ABB RobotStudio station: Robot_1530ID (task 1).rsstn

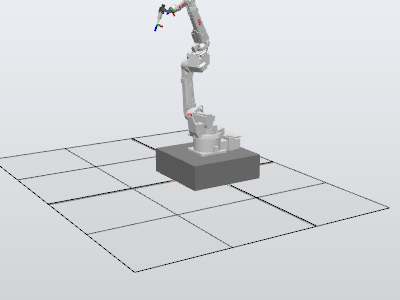
Station Robot_1520ID (frist class) (saved by RobotStudio 22.3.10141.1)
Controller Controller17, task T_ROB1: task frame (RAPID world) sits at (0, 0, 290) mm in the station
Controller Controller17
  mechanical unit ROB_1: IRB1520ID_4_150__02, 6 joints, base frame (0, 0, 0) mm
Layout (positions relative to the parent item):
  - IRB1520ID_4_150__02 [mechanism, from Robots\IRB1520ID_4_150_G_02.rslib] at (0, 0, 290) mm; joint values [0.1655, 0.0623, -1.1863, -0.1436, 1.6527, 0.0715] (rad or m)
  - Part_1_2 [part, from Robotics 7020\Cement Base.rslib] at (-450, -450, 0) mm
  - MyTool [mechanism, from Training Objects\myTool.rslib] at (497.52, 54.16, 1970.29) mm, rotated rx 180 ry 60 rz -180 deg
Attachment: MyTool is attached to IRB1520ID_4_150__02 / Link6
Targets, tools, work objects and paths stored in the station, written as RAPID:
! task T_ROB1
MODULE CalibData
  PERS tooldata MyTool:=[TRUE,[[31.792631019,0,229.638935148],[0.945518576,0,0.325568154,0]],[1,[0,0,1],[1,0,0,0],0,0,0]];
ENDMODULE

